FUNCTION_BLOCK Switch_Up_confirm (* Switching(demultiplexing) an event based on boolean input G *)
  (* Standard: 61499-2 *)
  (* Version 1.0, 2022-01-09, Fan *)
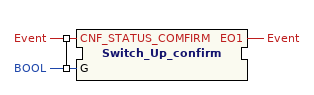
  EVENT_INPUT
    CNF_STATUS_COMFIRM WITH G;
  END_EVENT
  EVENT_OUTPUT
    EO1;
  END_EVENT
  VAR_INPUT
    G : BOOL;
  END_VAR
  EC_STATES
    START; (* Initial State *)
  END_STATES
END_FUNCTION_BLOCK
